// TIA Portal V19 export
FUNCTION_BLOCK "ButtonsSafe_LB114_FeedA01"   // FB99, LAD
TITLE = LB114 SAFE BUTTONS (@ Loop 1 / Rollformer entry) used for feed Area 01 material
// stored: MemoryReserve 100, SetENOAutomatically false
   VAR_INPUT
      Reset_OthersPBs_Activation_IN : Bool := FALSE;
   END_VAR
   VAR_OUTPUT
      Reset_OthersPBs_Activation_OUT : Bool;
   END_VAR
   VAR
      i : Int;
      iOperation : Int;
      iConcurrentOperation : Int;
      SettingWriteDone : Bool;
      PbPanel : "Buttons2Hands";
      PB : Struct
         ResetAlarms : Bool;
         Straightner_Fwd : Bool;
         Straightner_Bwd : Bool;
      END_STRUCT;
   END_VAR
   VAR CONSTANT
      ITEMS : Int := 2;
      STRAIGHTNER_FWD : Int := 1;
      STRAIGHTNER_BWD : Int := 2;
   END_VAR
BEGIN

REGION Network 1 (SCL): Interlocks between operations selected
   IF "Area01".AreaInterface.ManOneShot THEN
       #SettingWriteDone := FALSE;
   END_IF;

   // Interblocco tra operazioni
   // 
   IF NOT #SettingWriteDone THEN
       #SettingWriteDone := TRUE;

       FOR #iOperation := 1 TO #ITEMS DO
           FOR #iConcurrentOperation := 1 TO #ITEMS DO
               #PbPanel.Enables[#iOperation, #iConcurrentOperation] := FALSE;
           END_FOR;
       END_FOR;



   END_IF;
END_REGION

REGION Network 2 (SCL): Buttons for Op selection

   #PbPanel.Buttons[STRAIGHTNER_FWD] := "LB114_Straightener_Pb_Fwd";
   #PbPanel.Buttons[STRAIGHTNER_BWD] := "LB114_Straightener_Pb_Bwd";
END_REGION

REGION Network 3 (SCL): Operation enable

   #PbPanel.OpEnabled[STRAIGHTNER_FWD] := "Straightener".COut.Feed.Fwd_CheckNext;
   #PbPanel.OpEnabled[STRAIGHTNER_BWD] := "Straightener".COut.Feed.Bwd_CheckNext;
END_REGION

REGION Network 4 (SCL): Operation running

   #PbPanel.OpRunning[STRAIGHTNER_FWD] := "Straightener".COut.Feed.VelFwd_Running OR "Straightener".COut.Feed.PosFwd_Running;
   #PbPanel.OpRunning[STRAIGHTNER_BWD] := "Straightener".COut.Feed.VelBwd_Running OR "Straightener".COut.Feed.PosBwd_Running;
END_REGION

REGION Network 5 (SCL): Operation done

   #PbPanel.OpDone[STRAIGHTNER_FWD] := FALSE;
   #PbPanel.OpDone[STRAIGHTNER_BWD] := FALSE;
END_REGION

REGION Network 6: Main
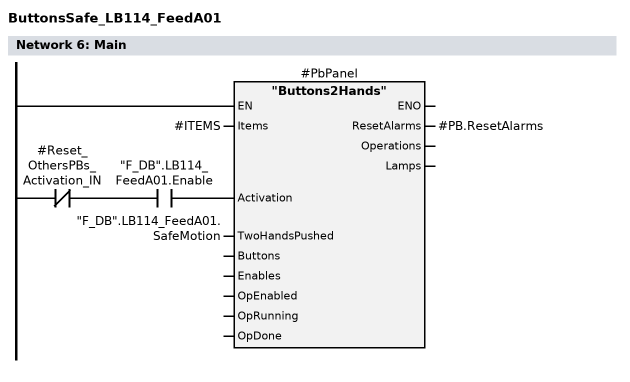
   RUNG wire#powerrail
      #PbPanel(Activation := wire#w1, Items := #ITEMS, TwoHandsPushed := "F_DB".LB114_FeedA01.SafeMotion, Buttons :=, Enables :=, OpEnabled :=, OpRunning :=, OpDone :=, ResetAlarms => #PB.ResetAlarms, Operations =>, Lamps =>)
   END_RUNG
   RUNG wire#powerrail
      I_Contact( #Reset_OthersPBs_Activation_IN )
      Contact( "F_DB".LB114_FeedA01.Enable )
   END_RUNG wire#w1
   // the same network as SCL:
   #PbPanel(Items := #ITEMS,   // "Buttons2Hands"
            Activation := NOT #Reset_OthersPBs_Activation_IN AND "F_DB".LB114_FeedA01.Enable,
            TwoHandsPushed := "F_DB".LB114_FeedA01.SafeMotion,
            ResetAlarms => #PB.ResetAlarms);
END_REGION

REGION Network 7 (SCL): Safe Buttons

   #PB.Straightner_Fwd := #PbPanel.Operations[STRAIGHTNER_FWD];
   #PB.Straightner_Bwd := #PbPanel.Operations[STRAIGHTNER_BWD];
END_REGION

REGION Network 8 (SCL): Lamp selection

   "LB114_Straightener_Lp_Fwd" := #PbPanel.Lamps[STRAIGHTNER_FWD];
   "LB114_Straightener_Lp_Bwd" := #PbPanel.Lamps[STRAIGHTNER_BWD];
END_REGION

REGION Network 9 (SCL): Reset others safe push buttons activation / execution
   #Reset_OthersPBs_Activation_OUT := FALSE;

   FOR #i := 1 TO #ITEMS DO

       IF #PbPanel.Buttons[#i] OR #PbPanel.Operations[#i] THEN
           #Reset_OthersPBs_Activation_OUT := TRUE;
           EXIT;
       END_IF;

   END_FOR;
END_REGION

REGION Network 10: >
END_REGION

REGION Network 11: >
END_REGION

REGION Network 12: >
END_REGION
END_FUNCTION_BLOCK
